(*Provides various mathematical functions*)
PROGRAM Math
VAR
END_VAR

(* 
    Time-compensated smoothing coefficient. 
    Alpha = 1 - (1 - B)^dt
*)
METHOD ExptDecay : LREAL
VAR_INPUT
    rBlendFactor : LREAL;   // In [0, 1] — how fast to blend toward input
    rDeltaTime   : LREAL := 0.01;   // In seconds
END_VAR
rBlendFactor := LIMIT(0.0, rBlendFactor, 1.0);
rDeltaTime   := MAX(rDeltaTime, 0.0);
ExptDecay := LIMIT(0.0, 1.0 - EXPT(1.0 - rBlendFactor, rDeltaTime), 1.0);
END_METHOD

(*
Allows for value scalling.
Returns 0 when rMaxX - rMinX = 0.
*)
METHOD LinearScale : LREAL
VAR_INPUT
	rX				: LREAL;
	rMinX			: LREAL;
	rMaxX			: LREAL;
	rMinY			: LREAL := 0;
	rMaxY			: LREAL := 1;
END_VAR
VAR
	_rDnmtr			: LREAL := rMaxX - rMinX;
END_VAR
IF _rDnmtr <> 0 THEN
	LinearScale := rMinY + ((rX - rMinX)/_rDnmtr) * (rMaxY - rMinY);
END_IF
END_METHOD

(*
First-order low pass filter.
Yt = Xt * Coeff + Y(t-1) * (1- Coeff)
*)
METHOD LowPassFilter : LREAL
VAR_INPUT
	rX				: LREAL;
	rPrvY			: LREAL;
	
	rCoefficient	: LREAL;
END_VAR
LowPassFilter := rX * rCoefficient + rPrvY * (1 - rCoefficient);
END_METHOD

(*
Generates random number every time is called.
*)
METHOD Random : LREAL
VAR_STAT
	_nSeed		: INT;
END_VAR
VAR
	_drand		: Tc2_System.DRAND;
END_VAR
_drand(Seed := _nSeed, Num => Random);
_nSeed := _nSeed + 1;
END_METHOD

END_PROGRAM

(* stored: Version 1.1.0.1
   POU Math: Id {76db6186-827d-4be6-8551-4ecec23c6cd1}, SpecialFunc None
   Method ExptDecay: Id {e059c742-3011-40a4-ba84-db0f8f8c97cf}
   Method LinearScale: Id {37fc285e-354d-4811-9875-fb9578429fc0}
   Method LowPassFilter: Id {54dd59a2-6c09-4c12-9961-65f71218b6f9}
   Method Random: Id {8fa98490-891b-4c1e-b9e9-80fb0f11e0b4} *)
